// TIA Portal V15.1 export
// export: Created 2024-05-17T05:38:31.1004631Z, ExportSetting WithDefaults, DisplayName Totally Integrated Automation Portal, DisplayVersion V15.1 Update 5, DisplayName TIA Portal Openness, DisplayVersion V15.1 Update 5, DisplayName SINAMICS Startdrive Advanced, DisplayVersion V15.1, DisplayName G130, G150, S120, S150, SINAMICS MV, S210, DisplayVersion V15.1, DisplayName G110M, G120, G120C, G120D, G120P, DisplayVersion V15.1, DisplayName STEP 7 Professional, DisplayVersion V15.1 Update 5, DisplayName STEP 7 Safety, DisplayVersion V15.1, DisplayName WinCC Professional, DisplayVersion V15.1 Update 5, DisplayName SIMATIC Visualization Architect, DisplayVersion V15.1
FUNCTION_BLOCK "LProductionMode"   // FB1003, FBD
TITLE = LProductionMode
{ S7_Optimized_Access := 'FALSE' }
AUTHOR : VCC
FAMILY : Control
NAME : ProdMode
VERSION : 1.0
// ================================================================================
// This module handles all production modes for a modezone. The production modes 
// are Bypass, Empty Station, Simulation with/without part, Maintenance, Cycle 
// Stop and Production Stop.
// ================================================================================
// stored: AutoNumber false, IsIECCheckEnabled false, SetENOAutomatically False, UDAEnableTagReadback false
   VAR_INPUT
      I_BypassStartCond { ExternalAccessible := 'False'; ExternalVisible := 'False'; ExternalWritable := 'False'} : Bool;   // Start condition for Bypass mode
      I_ExtBypassReq { ExternalAccessible := 'False'; ExternalVisible := 'False'; ExternalWritable := 'False'} : Bool;   // External bypass request
      I_EmptyStnReached { ExternalAccessible := 'False'; ExternalVisible := 'False'; ExternalWritable := 'False'} : Bool;   // Empty station reached
      I_ExtEmptyStnReq { ExternalAccessible := 'False'; ExternalVisible := 'False'; ExternalWritable := 'False'} : Bool;   // External Empty station request
      I_SimWithPartStartCond { ExternalAccessible := 'False'; ExternalVisible := 'False'; ExternalWritable := 'False'} : Bool;   // Start condition for Simulation with part mode
      I_ExtSimWithPartReq { ExternalAccessible := 'False'; ExternalVisible := 'False'; ExternalWritable := 'False'} : Bool;   // External Simulation with part request
      I_SimWithoutPartStartCon { ExternalAccessible := 'False'; ExternalVisible := 'False'; ExternalWritable := 'False'} : Bool;   // Start condition for Simulation without part mode
      I_ExtSimWithoutPartReq { ExternalAccessible := 'False'; ExternalVisible := 'False'; ExternalWritable := 'False'} : Bool;   // External Simulation without part request
      I_MaintStartCond { ExternalAccessible := 'False'; ExternalVisible := 'False'; ExternalWritable := 'False'} : Bool;   // Start condition for maintenance mode
      I_ExtMaintReq { ExternalAccessible := 'False'; ExternalVisible := 'False'; ExternalWritable := 'False'} : Bool;   // External Maintenance request
      I_MaintReached { ExternalAccessible := 'False'; ExternalVisible := 'False'; ExternalWritable := 'False'} : Bool;   // Maintenance reached
      I_CycleStpBeforeReached { ExternalAccessible := 'False'; ExternalVisible := 'False'; ExternalWritable := 'False'} : Bool;   // Cycle stop before work reached
      I_ExtCycleStpBeforeReq { ExternalAccessible := 'False'; ExternalVisible := 'False'; ExternalWritable := 'False'} : Bool;   // External Cycle stop before work request
      I_CycleStpAfterReached { ExternalAccessible := 'False'; ExternalVisible := 'False'; ExternalWritable := 'False'} : Bool;   // Cycle stop after work reached
      I_ExtCycleStpAfterReq { ExternalAccessible := 'False'; ExternalVisible := 'False'; ExternalWritable := 'False'} : Bool;   // External Cycle stop after work request
      I_ProdStpReached { ExternalAccessible := 'False'; ExternalVisible := 'False'; ExternalWritable := 'False'} : Bool;   // Production mode reached
      I_ExtProdStpReq { ExternalAccessible := 'False'; ExternalVisible := 'False'; ExternalWritable := 'False'} : Bool;   // External production stop request
      I_AlarmResetPB { ExternalAccessible := 'False'; ExternalVisible := 'False'; ExternalWritable := 'False'} : Bool;   // Alarm reset pushbutton is activated
   END_VAR
   VAR_OUTPUT
      O_ProductionMode { ExternalAccessible := 'False'; ExternalVisible := 'False'; ExternalWritable := 'False'} : Word;   // Prodution Modes
      O_BypassModeSel { ExternalAccessible := 'False'; ExternalVisible := 'False'; ExternalWritable := 'False'} : Bool;   // Bypass mode selected
      O_BypassMode { ExternalAccessible := 'False'; ExternalVisible := 'False'; ExternalWritable := 'False'} : Bool;   // Bypass mode active
      O_EmptyStnModeSel { ExternalAccessible := 'False'; ExternalVisible := 'False'; ExternalWritable := 'False'} : Bool;   // Empty station mode selected
      O_EmptyStnMode { ExternalAccessible := 'False'; ExternalVisible := 'False'; ExternalWritable := 'False'} : Bool;   // Empty station mode active
      O_SimWithPartModeSel { ExternalAccessible := 'False'; ExternalVisible := 'False'; ExternalWritable := 'False'} : Bool;   // Simulation with part mode selected
      O_SimWithPartMode { ExternalAccessible := 'False'; ExternalVisible := 'False'; ExternalWritable := 'False'} : Bool;   // Simulation with part mode active
      O_SimWithoutPartModeSel { ExternalAccessible := 'False'; ExternalVisible := 'False'; ExternalWritable := 'False'} : Bool;   // Simulation without part mode selcted
      O_SimWithoutPartMode { ExternalAccessible := 'False'; ExternalVisible := 'False'; ExternalWritable := 'False'} : Bool;   // Simulation without part mode active
      O_MaintModeSel { ExternalAccessible := 'False'; ExternalVisible := 'False'; ExternalWritable := 'False'} : Bool;   // Maintenance mode selected
      O_MaintMode { ExternalAccessible := 'False'; ExternalVisible := 'False'; ExternalWritable := 'False'} : Bool;   // Maintenance mode active
      O_CycleStpBeforeModeSel { ExternalAccessible := 'False'; ExternalVisible := 'False'; ExternalWritable := 'False'} : Bool;   // Cycle stop before mode selected
      O_CycleStpBeforeMode { ExternalAccessible := 'False'; ExternalVisible := 'False'; ExternalWritable := 'False'} : Bool;   // Cycle stop before mode active
      O_CycleStpAfterModeSel { ExternalAccessible := 'False'; ExternalVisible := 'False'; ExternalWritable := 'False'} : Bool;   // Cycle stop after mode selected
      O_CycleStpAfterMode { ExternalAccessible := 'False'; ExternalVisible := 'False'; ExternalWritable := 'False'} : Bool;   // Cycle stop after mode active
      O_ProdStpModeSel { ExternalAccessible := 'False'; ExternalVisible := 'False'; ExternalWritable := 'False'} : Bool;   // Production mode selected
      O_ProdStpMode { ExternalAccessible := 'False'; ExternalVisible := 'False'; ExternalWritable := 'False'} : Bool;   // Production mode active
      O_AnyProdModeSel { ExternalAccessible := 'False'; ExternalVisible := 'False'; ExternalWritable := 'False'} : Bool;   // Any production mode selected
      O_AnyProdModeActive { ExternalAccessible := 'False'; ExternalVisible := 'False'; ExternalWritable := 'False'} : Bool;   // Any production mode active
      O_AlarmABCondition { ExternalAccessible := 'False'; ExternalVisible := 'False'; ExternalWritable := 'False'} : Bool;   // Alarm AB condition
      O_AlarmA { ExternalAccessible := 'False'; ExternalVisible := 'False'; ExternalWritable := 'False'} : Bool;   // Alarms A
      O_AlarmB { ExternalAccessible := 'False'; ExternalVisible := 'False'; ExternalWritable := 'False'} : Bool;   // Alarms B
      O_AlarmC { ExternalAccessible := 'False'; ExternalVisible := 'False'; ExternalWritable := 'False'} : Bool;   // Alarms C
      O_AlarmD { ExternalAccessible := 'False'; ExternalVisible := 'False'; ExternalWritable := 'False'} : Bool;   // Alarms D
      H_AlarmWord { ExternalAccessible := 'False'; ExternalVisible := 'False'; ExternalWritable := 'False'} : DWord;   // Alarm Word
   END_VAR
   VAR_IN_OUT
      IO_Modes : "Modes";
   END_VAR
   VAR DB_SPECIFIC
      AB_SimWithPartAlm { ExternalAccessible := 'False'; ExternalVisible := 'False'; ExternalWritable := 'False'} : Bool;   // Condition missing for simulation with part
      AB_SimWithoutPartAlm { ExternalAccessible := 'False'; ExternalVisible := 'False'; ExternalWritable := 'False'} : Bool;   // Condition missing for simulation without part
      AD_EmptyStnSelected { ExternalAccessible := 'False'; ExternalVisible := 'False'; ExternalWritable := 'False'} : Bool;   // Empty station is selected
      AD_BypassSelected { ExternalAccessible := 'False'; ExternalVisible := 'False'; ExternalWritable := 'False'} : Bool;   // Bypass is selected
      AD_SimWithPartSelected { ExternalAccessible := 'False'; ExternalVisible := 'False'; ExternalWritable := 'False'} : Bool;   // Simulation with part is selected
      AD_SimWithoutPartSel { ExternalAccessible := 'False'; ExternalVisible := 'False'; ExternalWritable := 'False'} : Bool;   // Simulation without part is selected
      AD_MaintSelected { ExternalAccessible := 'False'; ExternalVisible := 'False'; ExternalWritable := 'False'} : Bool;   // Maintenance is selected
      AD_ProdStpSelected { ExternalAccessible := 'False'; ExternalVisible := 'False'; ExternalWritable := 'False'} : Bool;   // Production stop is selected
      AD_CycleStpBeforeSel { ExternalAccessible := 'False'; ExternalVisible := 'False'; ExternalWritable := 'False'} : Bool;   // Cycle stop before is selected
      AD_CycleStpAfterSelected { ExternalAccessible := 'False'; ExternalVisible := 'False'; ExternalWritable := 'False'} : Bool;   // Cycle stop after is selected
      H_HMIProdModeCmd : Word;   // Production mode commands from HMI
      H_Anim : Word;   // Animation
      H_Anim2 : Word;   // Animation word 2
      SimWithPartAlmCond { ExternalAccessible := 'False'; ExternalVisible := 'False'; ExternalWritable := 'False'} : Bool;   // Alarm condition for Simulation with part
      SimWithoutPartAlmCond { ExternalAccessible := 'False'; ExternalVisible := 'False'; ExternalWritable := 'False'} : Bool;   // Alarm condition for Simulation without part
      HMIBypassReq { ExternalAccessible := 'False'; ExternalVisible := 'False'; ExternalWritable := 'False'} : Bool;   // Bypass selected on HMI
      HMIEmptyStnReq { ExternalAccessible := 'False'; ExternalVisible := 'False'; ExternalWritable := 'False'} : Bool;   // Empty station selected on HMI
      HMISimWithPartReq { ExternalAccessible := 'False'; ExternalVisible := 'False'; ExternalWritable := 'False'} : Bool;   // Simulation with part selected on HMI
      HMISimWithoutPartReq { ExternalAccessible := 'False'; ExternalVisible := 'False'; ExternalWritable := 'False'} : Bool;   // Simulation without part selected on HMI
      HMIMaintReq { ExternalAccessible := 'False'; ExternalVisible := 'False'; ExternalWritable := 'False'} : Bool;   // Maintenance selected on HMI
      HMICycleStpBeforeReq { ExternalAccessible := 'False'; ExternalVisible := 'False'; ExternalWritable := 'False'} : Bool;   // Cycle stop before work selected on HMI
      HMICycleStpAfterReq { ExternalAccessible := 'False'; ExternalVisible := 'False'; ExternalWritable := 'False'} : Bool;   // Cycle stop after work selected on HMI
      HMIProdStpReq { ExternalAccessible := 'False'; ExternalVisible := 'False'; ExternalWritable := 'False'} : Bool;   // Production mode selected on HMI
      EmptyStnActive { ExternalAccessible := 'False'; ExternalVisible := 'False'; ExternalWritable := 'False'} : Bool;   // Empty station is active
      BypassActive { ExternalAccessible := 'False'; ExternalVisible := 'False'; ExternalWritable := 'False'} : Bool;   // Bypass is active
      SimWithPartActive { ExternalAccessible := 'False'; ExternalVisible := 'False'; ExternalWritable := 'False'} : Bool;   // Simulation with part is active
      SimWithoutPartActive { ExternalAccessible := 'False'; ExternalVisible := 'False'; ExternalWritable := 'False'} : Bool;   // Simulation without part is active
      SimDeactivate { ExternalAccessible := 'False'; ExternalVisible := 'False'; ExternalWritable := 'False'} : Bool;   // Deactivate simulation
      MaintActive { ExternalAccessible := 'False'; ExternalVisible := 'False'; ExternalWritable := 'False'} : Bool;   // Maintenance is active
      ProdStpActive { ExternalAccessible := 'False'; ExternalVisible := 'False'; ExternalWritable := 'False'} : Bool;   // Production stop is active
      CycleStpBeforeActive { ExternalAccessible := 'False'; ExternalVisible := 'False'; ExternalWritable := 'False'} : Bool;   // Cycle stop before is active
      CycleStpAfterActive { ExternalAccessible := 'False'; ExternalVisible := 'False'; ExternalWritable := 'False'} : Bool;   // Cycle stop after is active
      PulseSimWithPartSel { ExternalAccessible := 'False'; ExternalVisible := 'False'; ExternalWritable := 'False'} : Bool;   // Pulse simulation with part selected
      PulseSimWithoutPartSel { ExternalAccessible := 'False'; ExternalVisible := 'False'; ExternalWritable := 'False'} : Bool;   // Pulse simulation without part selected
      TmpMaintReqOn { ExternalAccessible := 'False'; ExternalVisible := 'False'; ExternalWritable := 'False'} : Bool;   // Temporary request on
      TmpBypassReqOn { ExternalAccessible := 'False'; ExternalVisible := 'False'; ExternalWritable := 'False'} : Bool;   // Temporary request on
      TmpEmptyStnReqOn { ExternalAccessible := 'False'; ExternalVisible := 'False'; ExternalWritable := 'False'} : Bool;   // Temporary request on
      TmpProdStpReqOn { ExternalAccessible := 'False'; ExternalVisible := 'False'; ExternalWritable := 'False'} : Bool;   // Temporary request on
      AlarmA { ExternalAccessible := 'False'; ExternalVisible := 'False'; ExternalWritable := 'False'} : Bool;   // Alarm A active in the FB
      AlarmB { ExternalAccessible := 'False'; ExternalVisible := 'False'; ExternalWritable := 'False'} : Bool;   // Alarm B active in the FB
      AlarmC { ExternalAccessible := 'False'; ExternalVisible := 'False'; ExternalWritable := 'False'} : Bool;   // Alarm C active in the FB
      AlarmD { ExternalAccessible := 'False'; ExternalVisible := 'False'; ExternalWritable := 'False'} : Bool;   // Alarm D active in the FB
      TmpSimWithoutPartReqOn { ExternalAccessible := 'False'; ExternalVisible := 'False'; ExternalWritable := 'False'} : Bool;   // Temporary request on
      TmpSimWithPartReqOn { ExternalAccessible := 'False'; ExternalVisible := 'False'; ExternalWritable := 'False'} : Bool;   // Temporary request on
   END_VAR
   VAR
      ToggleBypassReq { ExternalAccessible := 'False'; ExternalVisible := 'False'; ExternalWritable := 'False'; S7_SetPoint := 'True'} : "LToggle";
      ToggleEmptyStnReq { ExternalAccessible := 'False'; ExternalVisible := 'False'; ExternalWritable := 'False'; S7_SetPoint := 'True'} : "LToggle";
      ToggleSimWithPartReq { ExternalAccessible := 'False'; ExternalVisible := 'False'; ExternalWritable := 'False'; S7_SetPoint := 'True'} : "LToggle";
      ToggleMaintReq { ExternalAccessible := 'False'; ExternalVisible := 'False'; ExternalWritable := 'False'; S7_SetPoint := 'True'} : "LToggle";
      ToggleCycleStpBeforeReq { ExternalAccessible := 'False'; ExternalVisible := 'False'; ExternalWritable := 'False'; S7_SetPoint := 'True'} : "LToggle";
      ToggleCycleStpAfterReq { ExternalAccessible := 'False'; ExternalVisible := 'False'; ExternalWritable := 'False'; S7_SetPoint := 'True'} : "LToggle";
      ToggleProsStpReq { ExternalAccessible := 'False'; ExternalVisible := 'False'; ExternalWritable := 'False'; S7_SetPoint := 'True'} : "LToggle";
      ToggleSimWithoutPartReq { ExternalAccessible := 'False'; ExternalVisible := 'False'; ExternalWritable := 'False'; S7_SetPoint := 'True'} : "LToggle";
   END_VAR
   VAR_TEMP   // added for the SCL form of the ladder/FBD networks
      _w1 : Bool;
   END_VAR
BEGIN

REGION Network 1: **** 1 - Inputs **** Extract the production modes from HMI
   // Extract the production modes from HMI
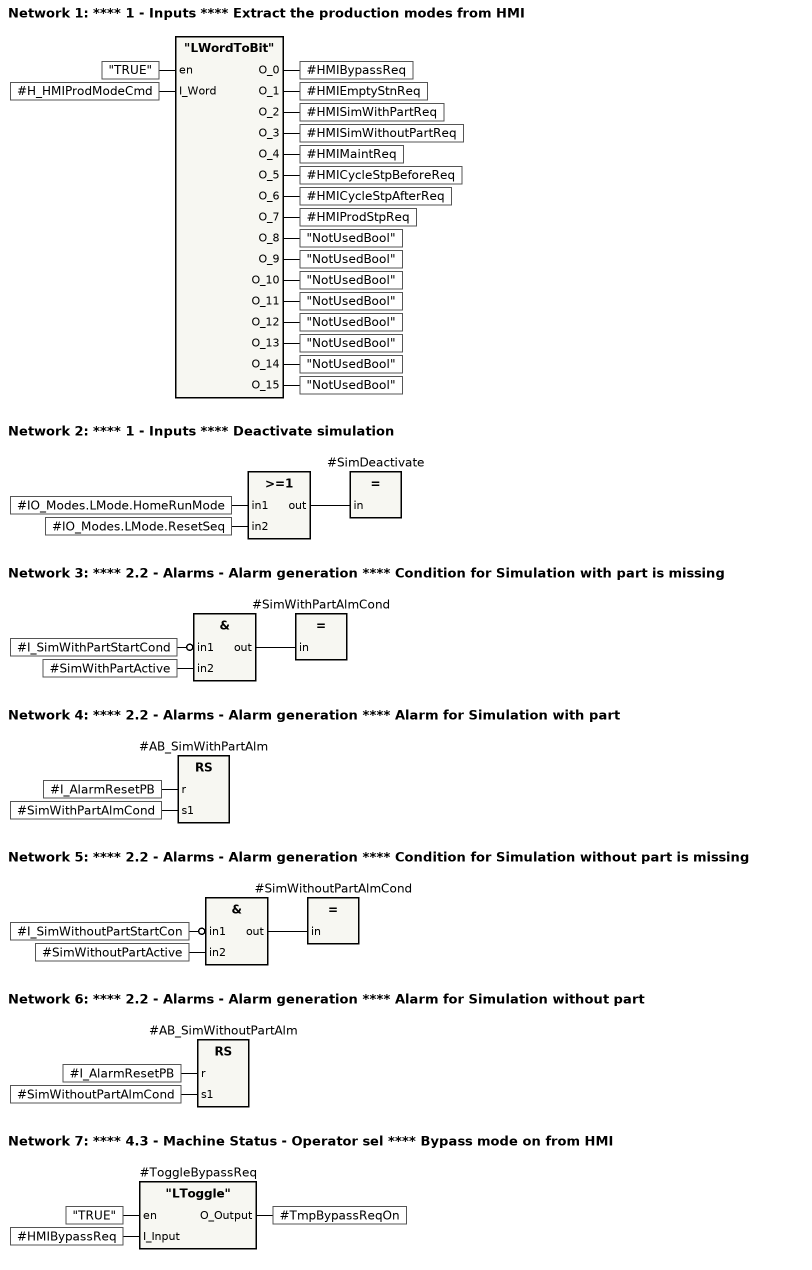
   IF "TRUE" THEN
       "LWordToBit"(I_Word := #H_HMIProdModeCmd,
                    O_0 => #HMIBypassReq,
                    O_1 => #HMIEmptyStnReq,
                    O_2 => #HMISimWithPartReq,
                    O_3 => #HMISimWithoutPartReq,
                    O_4 => #HMIMaintReq,
                    O_5 => #HMICycleStpBeforeReq,
                    O_6 => #HMICycleStpAfterReq,
                    O_7 => #HMIProdStpReq,
                    O_8 => "NotUsedBool",
                    O_9 => "NotUsedBool",
                    O_10 => "NotUsedBool",
                    O_11 => "NotUsedBool",
                    O_12 => "NotUsedBool",
                    O_13 => "NotUsedBool",
                    O_14 => "NotUsedBool",
                    O_15 => "NotUsedBool");
   END_IF;
END_REGION

REGION Network 2: **** 1 - Inputs **** Deactivate simulation
   #SimDeactivate := #IO_Modes.LMode.HomeRunMode OR #IO_Modes.LMode.ResetSeq;
END_REGION

REGION Network 3: **** 2.2 - Alarms - Alarm generation **** Condition for Simulation with part is missing
   // Condition for Simulation with part is missing
   #SimWithPartAlmCond := NOT #I_SimWithPartStartCond AND #SimWithPartActive;
END_REGION

REGION Network 4: **** 2.2 - Alarms - Alarm generation **** Alarm for Simulation with part
   // Alarm for Simulation with part
   IF #I_AlarmResetPB THEN
       #AB_SimWithPartAlm := FALSE;   // RS flip-flop
   END_IF;
   IF #SimWithPartAlmCond THEN #AB_SimWithPartAlm := TRUE; END_IF;
END_REGION

REGION Network 5: **** 2.2 - Alarms - Alarm generation **** Condition for Simulation without part is missing
   // Condition for Simulation without part is missing
   #SimWithoutPartAlmCond := NOT #I_SimWithoutPartStartCon AND #SimWithoutPartActive;
END_REGION

REGION Network 6: **** 2.2 - Alarms - Alarm generation **** Alarm for Simulation without part
   // Alarm for Simulation without part
   IF #I_AlarmResetPB THEN
       #AB_SimWithoutPartAlm := FALSE;   // RS flip-flop
   END_IF;
   IF #SimWithoutPartAlmCond THEN #AB_SimWithoutPartAlm := TRUE; END_IF;
END_REGION

REGION Network 7: **** 4.3 - Machine Status - Operator sel **** Bypass mode on from HMI
   // Bypass mode on from HMI
   IF "TRUE" THEN
       #ToggleBypassReq(I_Input := #HMIBypassReq, O_Output => #TmpBypassReqOn);   // "LToggle"
   END_IF;
END_REGION

REGION Network 8: **** 4.3 - Machine Status - Operator sel **** Bypass mode is selected
   // Bypass mode is selected
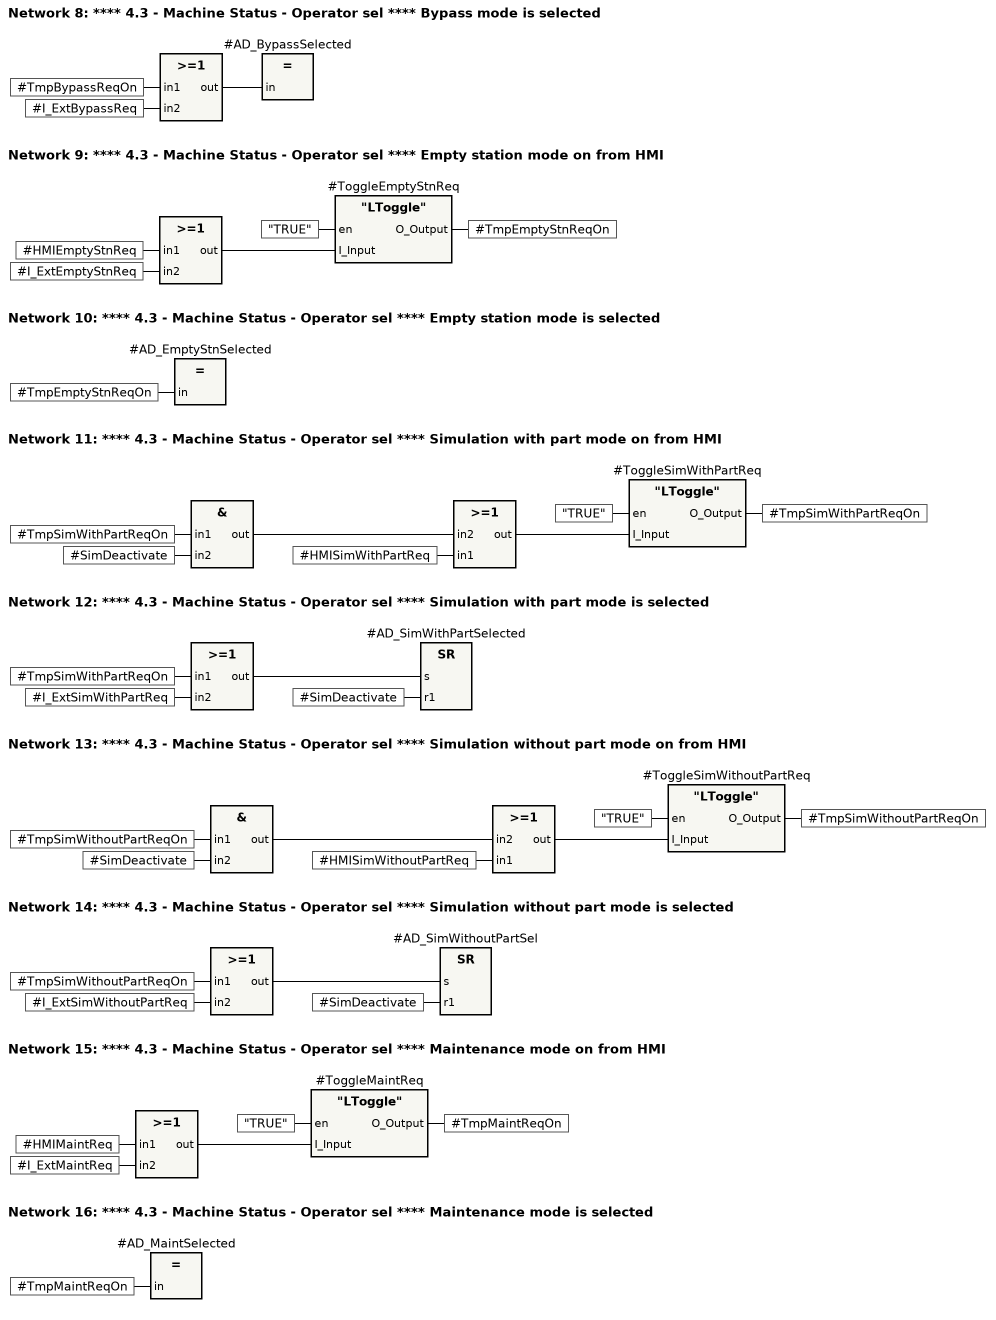
   #AD_BypassSelected := #TmpBypassReqOn OR #I_ExtBypassReq;
END_REGION

REGION Network 9: **** 4.3 - Machine Status - Operator sel **** Empty station mode on from HMI
   // Empty station mode on from HMI
   IF "TRUE" THEN
       #ToggleEmptyStnReq(I_Input := #HMIEmptyStnReq OR #I_ExtEmptyStnReq, O_Output => #TmpEmptyStnReqOn);   // "LToggle"
   END_IF;
END_REGION

REGION Network 10: **** 4.3 - Machine Status - Operator sel **** Empty station mode is selected
   // Empty station mode is selected
   #AD_EmptyStnSelected := #TmpEmptyStnReqOn;
END_REGION

REGION Network 11: **** 4.3 - Machine Status - Operator sel **** Simulation with part mode on from HMI
   // Simulation with part mode on from HMI
   IF "TRUE" THEN
       #ToggleSimWithPartReq(I_Input := (#TmpSimWithPartReqOn AND #SimDeactivate) OR #HMISimWithPartReq,   // "LToggle"
                             O_Output => #TmpSimWithPartReqOn);
   END_IF;
END_REGION

REGION Network 12: **** 4.3 - Machine Status - Operator sel **** Simulation with part mode is selected
   // Simulation with part mode is selected
   IF #TmpSimWithPartReqOn OR #I_ExtSimWithPartReq THEN
       #AD_SimWithPartSelected := TRUE;   // SR flip-flop
   END_IF;
   IF #SimDeactivate THEN #AD_SimWithPartSelected := FALSE; END_IF;
END_REGION

REGION Network 13: **** 4.3 - Machine Status - Operator sel **** Simulation without part mode on from HMI
   // Simulation without part mode on from HMI
   IF "TRUE" THEN
       #ToggleSimWithoutPartReq(I_Input := (#TmpSimWithoutPartReqOn AND #SimDeactivate) OR #HMISimWithoutPartReq,   // "LToggle"
                               O_Output => #TmpSimWithoutPartReqOn);
   END_IF;
END_REGION

REGION Network 14: **** 4.3 - Machine Status - Operator sel **** Simulation without part mode is selected
   // Simulation without part mode is selected
   IF #TmpSimWithoutPartReqOn OR #I_ExtSimWithoutPartReq THEN
       #AD_SimWithoutPartSel := TRUE;   // SR flip-flop
   END_IF;
   IF #SimDeactivate THEN #AD_SimWithoutPartSel := FALSE; END_IF;
END_REGION

REGION Network 15: **** 4.3 - Machine Status - Operator sel **** Maintenance mode on from HMI
   // Maintenance mode on from HMI
   IF "TRUE" THEN
       #ToggleMaintReq(I_Input := #HMIMaintReq OR #I_ExtMaintReq, O_Output => #TmpMaintReqOn);   // "LToggle"
   END_IF;
END_REGION

REGION Network 16: **** 4.3 - Machine Status - Operator sel **** Maintenance mode is selected
   // Maintenance mode is selected
   #AD_MaintSelected := #TmpMaintReqOn;
END_REGION

REGION Network 17: **** 4.3 - Machine Status - Operator sel **** Cycle stop before mode is selected
   // Cycle stop before mode is selected
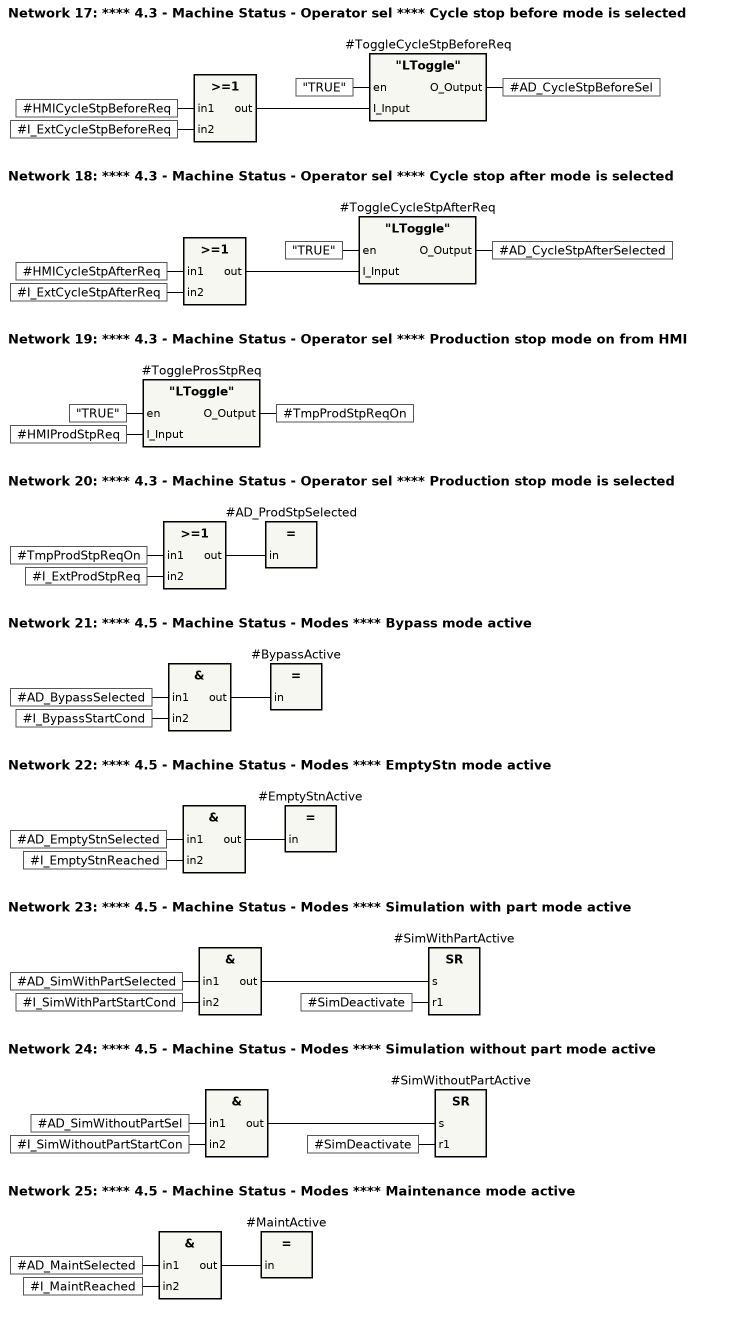
   IF "TRUE" THEN
       #ToggleCycleStpBeforeReq(I_Input := #HMICycleStpBeforeReq OR #I_ExtCycleStpBeforeReq,   // "LToggle"
                               O_Output => #AD_CycleStpBeforeSel);
   END_IF;
END_REGION

REGION Network 18: **** 4.3 - Machine Status - Operator sel **** Cycle stop after mode is selected
   // Cycle stop after mode is selected
   IF "TRUE" THEN
       #ToggleCycleStpAfterReq(I_Input := #HMICycleStpAfterReq OR #I_ExtCycleStpAfterReq,   // "LToggle"
                               O_Output => #AD_CycleStpAfterSelected);
   END_IF;
END_REGION

REGION Network 19: **** 4.3 - Machine Status - Operator sel **** Production stop mode on from HMI
   // Production stop mode on from HMI
   IF "TRUE" THEN
       #ToggleProsStpReq(I_Input := #HMIProdStpReq, O_Output => #TmpProdStpReqOn);   // "LToggle"
   END_IF;
END_REGION

REGION Network 20: **** 4.3 - Machine Status - Operator sel **** Production stop mode is selected
   // Production stop mode is selected
   #AD_ProdStpSelected := #TmpProdStpReqOn OR #I_ExtProdStpReq;
END_REGION

REGION Network 21: **** 4.5 - Machine Status - Modes **** Bypass mode active
   // Bypass mode active
   #BypassActive := #AD_BypassSelected AND #I_BypassStartCond;
END_REGION

REGION Network 22: **** 4.5 - Machine Status - Modes **** EmptyStn mode active
   // EmptyStn mode active
   #EmptyStnActive := #AD_EmptyStnSelected AND #I_EmptyStnReached;
END_REGION

REGION Network 23: **** 4.5 - Machine Status - Modes **** Simulation with part mode active
   // Simulation with part mode active
   IF #AD_SimWithPartSelected AND #I_SimWithPartStartCond THEN
       #SimWithPartActive := TRUE;   // SR flip-flop
   END_IF;
   IF #SimDeactivate THEN #SimWithPartActive := FALSE; END_IF;
END_REGION

REGION Network 24: **** 4.5 - Machine Status - Modes **** Simulation without part mode active
   // Simulation without part mode active
   IF #AD_SimWithoutPartSel AND #I_SimWithoutPartStartCon THEN
       #SimWithoutPartActive := TRUE;   // SR flip-flop
   END_IF;
   IF #SimDeactivate THEN #SimWithoutPartActive := FALSE; END_IF;
END_REGION

REGION Network 25: **** 4.5 - Machine Status - Modes **** Maintenance mode active
   // Maintenance mode active
   #MaintActive := #AD_MaintSelected AND #I_MaintReached;
END_REGION

REGION Network 26: **** 4.5 - Machine Status - Modes **** Cycle Stop Before mode active
   // Cycle Stop Before mode active
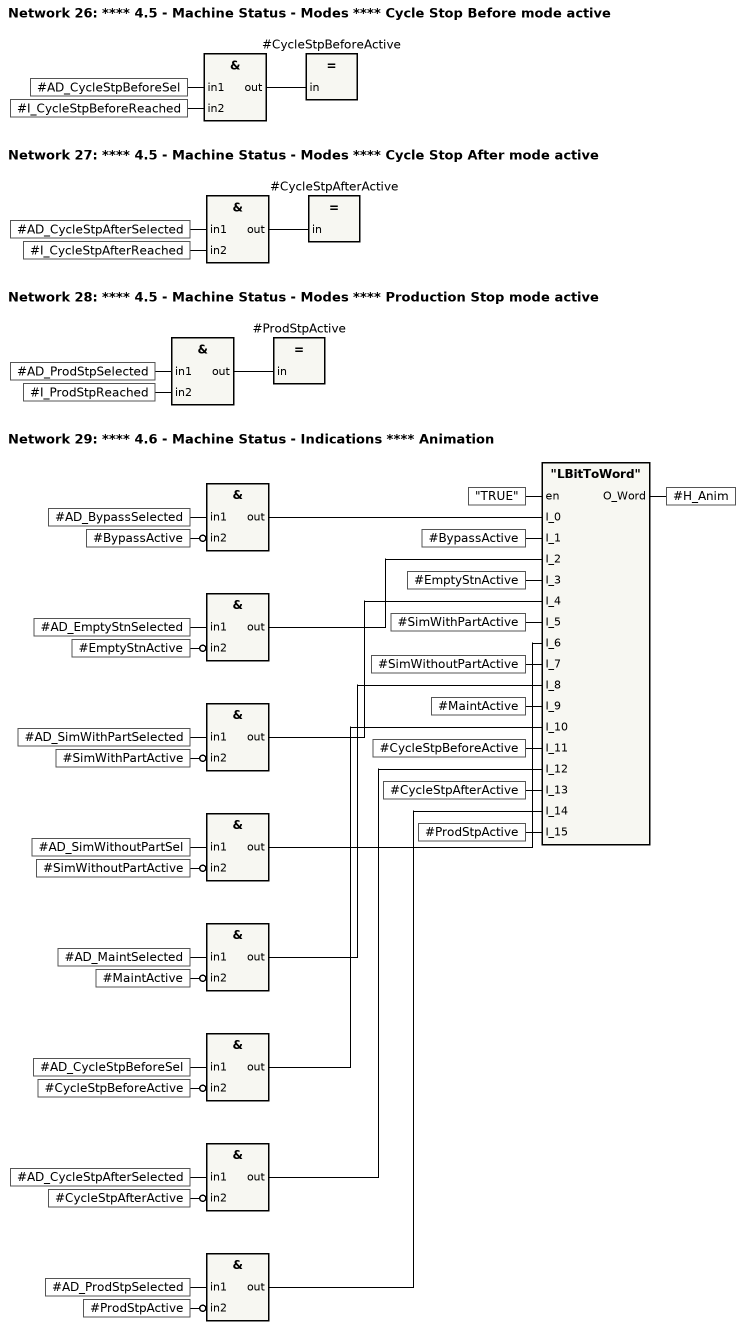
   #CycleStpBeforeActive := #AD_CycleStpBeforeSel AND #I_CycleStpBeforeReached;
END_REGION

REGION Network 27: **** 4.5 - Machine Status - Modes **** Cycle Stop After mode active
   // Cycle Stop After mode active
   #CycleStpAfterActive := #AD_CycleStpAfterSelected AND #I_CycleStpAfterReached;
END_REGION

REGION Network 28: **** 4.5 - Machine Status - Modes **** Production Stop mode active
   // Production Stop mode active
   #ProdStpActive := #AD_ProdStpSelected AND #I_ProdStpReached;
END_REGION

REGION Network 29: **** 4.6 - Machine Status - Indications **** Animation
   // Animation
   IF "TRUE" THEN
       "LBitToWord"(I_0 := #AD_BypassSelected AND NOT #BypassActive,
                    I_1 := #BypassActive,
                    I_2 := #AD_EmptyStnSelected AND NOT #EmptyStnActive,
                    I_3 := #EmptyStnActive,
                    I_4 := #AD_SimWithPartSelected AND NOT #SimWithPartActive,
                    I_5 := #SimWithPartActive,
                    I_6 := #AD_SimWithoutPartSel AND NOT #SimWithoutPartActive,
                    I_7 := #SimWithoutPartActive,
                    I_8 := #AD_MaintSelected AND NOT #MaintActive,
                    I_9 := #MaintActive,
                    I_10 := #AD_CycleStpBeforeSel AND NOT #CycleStpBeforeActive,
                    I_11 := #CycleStpBeforeActive,
                    I_12 := #AD_CycleStpAfterSelected AND NOT #CycleStpAfterActive,
                    I_13 := #CycleStpAfterActive,
                    I_14 := #AD_ProdStpSelected AND NOT #ProdStpActive,
                    I_15 := #ProdStpActive,
                    O_Word => #H_Anim);
   END_IF;
END_REGION

REGION Network 30: **** 4.6 - Machine Status - Indications **** Animation2
   // Animation word 2
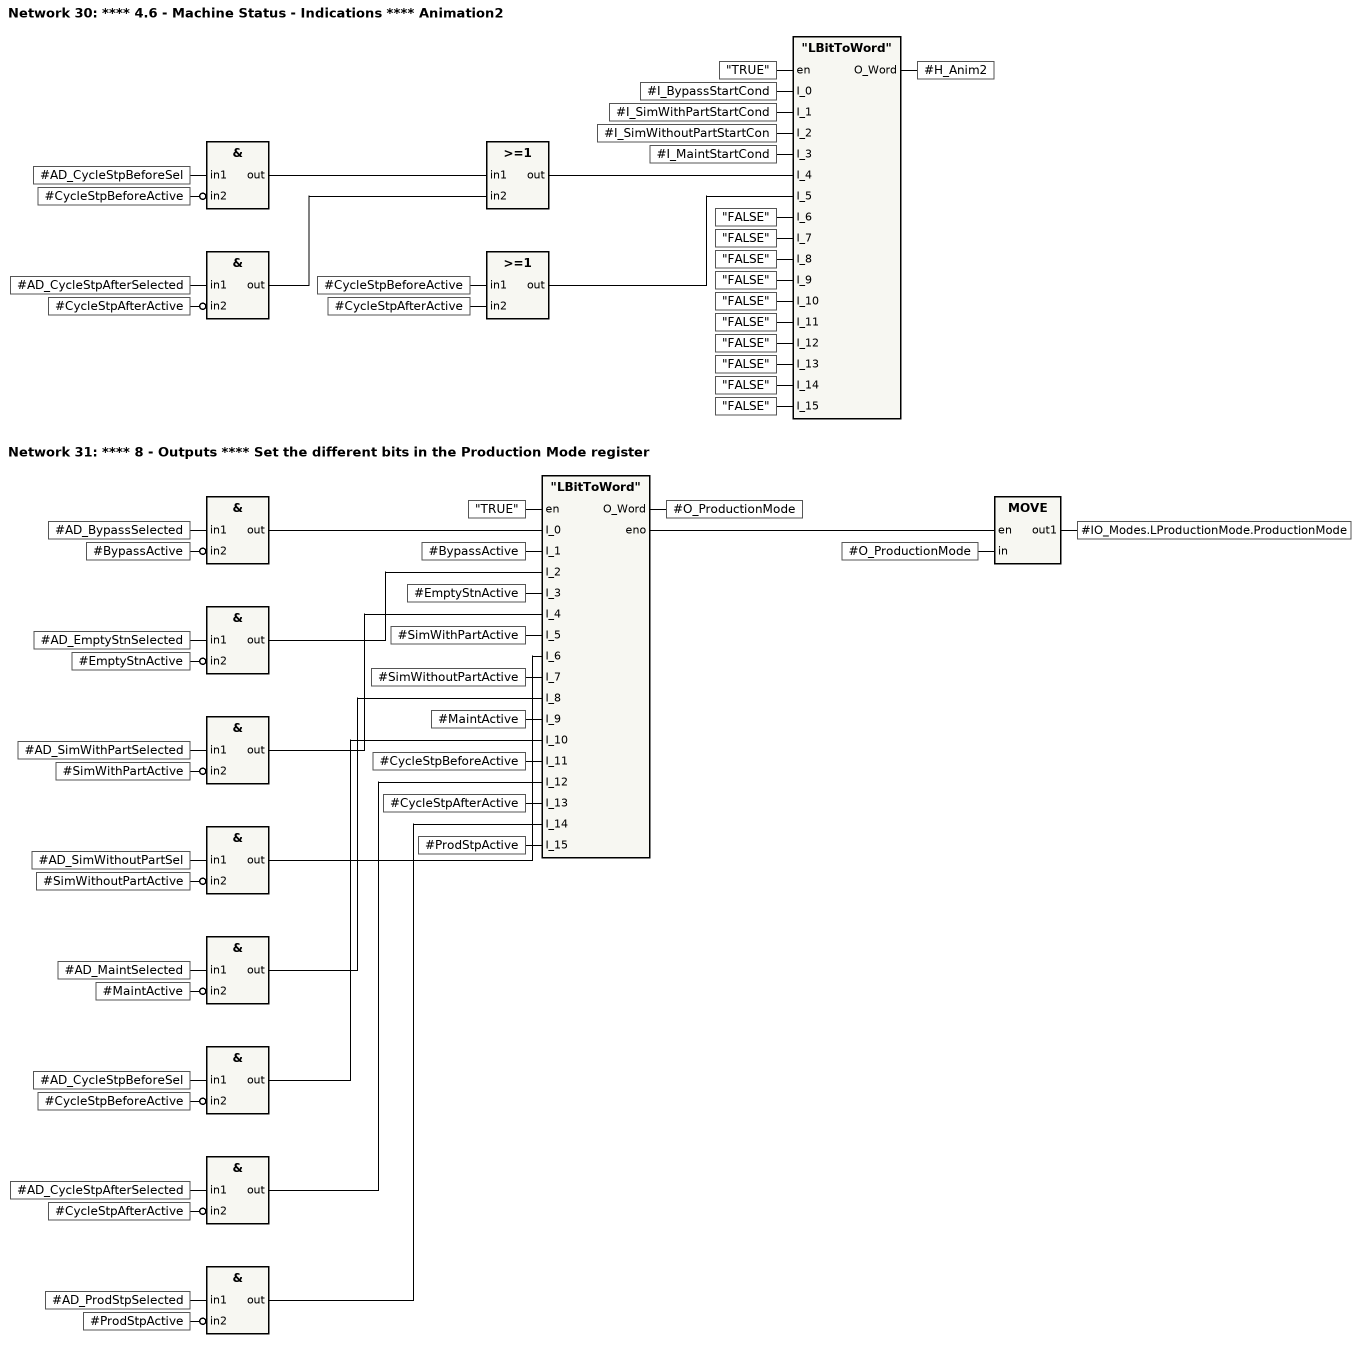
   IF "TRUE" THEN
       "LBitToWord"(I_0 := #I_BypassStartCond,
                    I_1 := #I_SimWithPartStartCond,
                    I_2 := #I_SimWithoutPartStartCon,
                    I_3 := #I_MaintStartCond,
                    I_4 := (#AD_CycleStpBeforeSel AND NOT #CycleStpBeforeActive) OR (#AD_CycleStpAfterSelected AND NOT #CycleStpAfterActive),
                    I_5 := #CycleStpBeforeActive OR #CycleStpAfterActive,
                    I_6 := "FALSE",
                    I_7 := "FALSE",
                    I_8 := "FALSE",
                    I_9 := "FALSE",
                    I_10 := "FALSE",
                    I_11 := "FALSE",
                    I_12 := "FALSE",
                    I_13 := "FALSE",
                    I_14 := "FALSE",
                    I_15 := "FALSE",
                    O_Word => #H_Anim2);
   END_IF;
END_REGION

REGION Network 31: **** 8 - Outputs **** Set the different bits in the Production Mode register
   // Set the different bits in the Production Mode register
   "LBitToWord"(EN := "TRUE",
                I_0 := #AD_BypassSelected AND NOT #BypassActive,
                I_1 := #BypassActive,
                I_2 := #AD_EmptyStnSelected AND NOT #EmptyStnActive,
                I_3 := #EmptyStnActive,
                I_4 := #AD_SimWithPartSelected AND NOT #SimWithPartActive,
                I_5 := #SimWithPartActive,
                I_6 := #AD_SimWithoutPartSel AND NOT #SimWithoutPartActive,
                I_7 := #SimWithoutPartActive,
                I_8 := #AD_MaintSelected AND NOT #MaintActive,
                I_9 := #MaintActive,
                I_10 := #AD_CycleStpBeforeSel AND NOT #CycleStpBeforeActive,
                I_11 := #CycleStpBeforeActive,
                I_12 := #AD_CycleStpAfterSelected AND NOT #CycleStpAfterActive,
                I_13 := #CycleStpAfterActive,
                I_14 := #AD_ProdStpSelected AND NOT #ProdStpActive,
                I_15 := #ProdStpActive,
                O_Word => #O_ProductionMode,
                ENO => #_w1);
   IF #_w1 THEN #IO_Modes.LProductionMode.ProductionMode := #O_ProductionMode; END_IF;
END_REGION

REGION Network 32: **** 8 - Outputs **** Bypass mode selected
   // Bypass mode selected
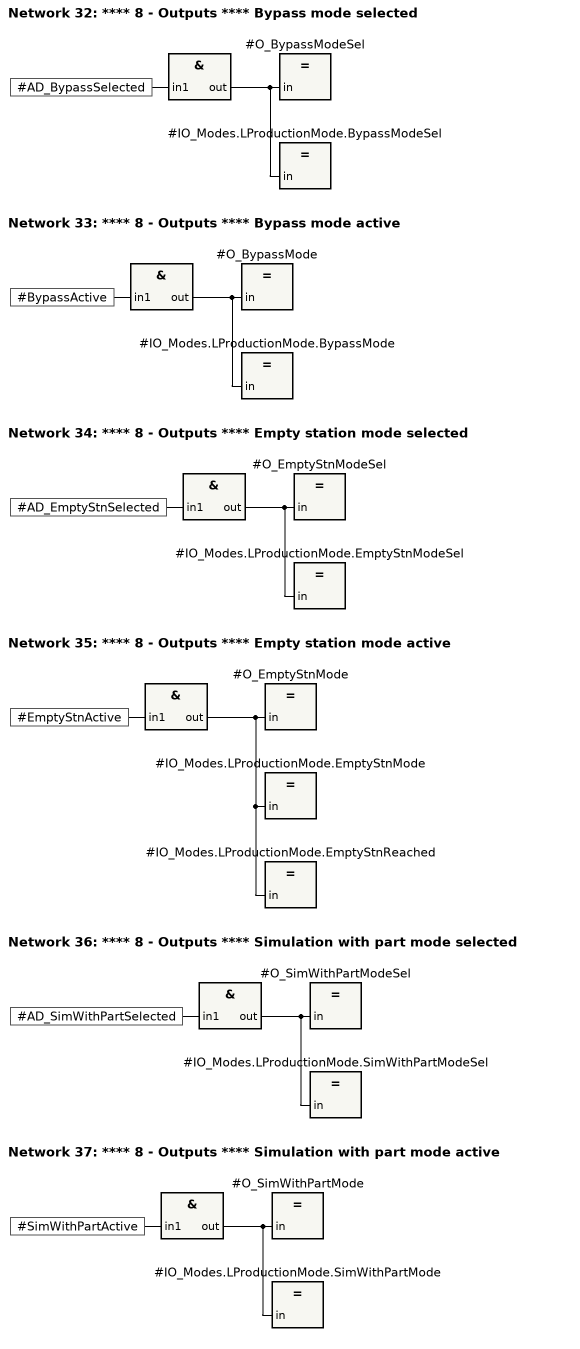
   #O_BypassModeSel := #AD_BypassSelected;
   #IO_Modes.LProductionMode.BypassModeSel := #AD_BypassSelected;
END_REGION

REGION Network 33: **** 8 - Outputs **** Bypass mode active
   // Bypass mode active
   #O_BypassMode := #BypassActive;
   #IO_Modes.LProductionMode.BypassMode := #BypassActive;
END_REGION

REGION Network 34: **** 8 - Outputs **** Empty station mode selected
   // Empty station mode selected
   #O_EmptyStnModeSel := #AD_EmptyStnSelected;
   #IO_Modes.LProductionMode.EmptyStnModeSel := #AD_EmptyStnSelected;
END_REGION

REGION Network 35: **** 8 - Outputs **** Empty station mode active
   // Empty station mode active
   #O_EmptyStnMode := #EmptyStnActive;
   #IO_Modes.LProductionMode.EmptyStnMode := #EmptyStnActive;
   #IO_Modes.LProductionMode.EmptyStnReached := #EmptyStnActive;
END_REGION

REGION Network 36: **** 8 - Outputs **** Simulation with part mode selected
   // Simulation with part mode selected
   #O_SimWithPartModeSel := #AD_SimWithPartSelected;
   #IO_Modes.LProductionMode.SimWithPartModeSel := #AD_SimWithPartSelected;
END_REGION

REGION Network 37: **** 8 - Outputs **** Simulation with part mode active
   // Simulation with part mode active
   #O_SimWithPartMode := #SimWithPartActive;
   #IO_Modes.LProductionMode.SimWithPartMode := #SimWithPartActive;
END_REGION

REGION Network 38: **** 8 - Outputs **** Simulation without part mode selected
   // Simulation without part mode selected
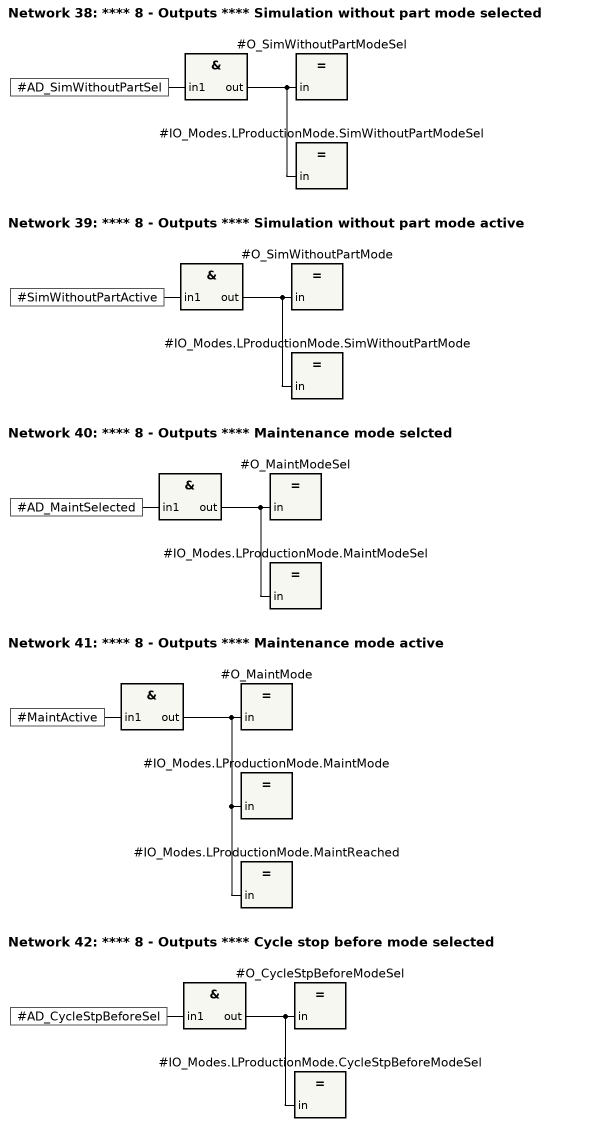
   #O_SimWithoutPartModeSel := #AD_SimWithoutPartSel;
   #IO_Modes.LProductionMode.SimWithoutPartModeSel := #AD_SimWithoutPartSel;
END_REGION

REGION Network 39: **** 8 - Outputs **** Simulation without part mode active
   // Simulation without part mode active
   #O_SimWithoutPartMode := #SimWithoutPartActive;
   #IO_Modes.LProductionMode.SimWithoutPartMode := #SimWithoutPartActive;
END_REGION

REGION Network 40: **** 8 - Outputs **** Maintenance mode selcted
   // Maintenance mode selcted
   #O_MaintModeSel := #AD_MaintSelected;
   #IO_Modes.LProductionMode.MaintModeSel := #AD_MaintSelected;
END_REGION

REGION Network 41: **** 8 - Outputs **** Maintenance mode active
   // Maintenance mode active
   #O_MaintMode := #MaintActive;
   #IO_Modes.LProductionMode.MaintMode := #MaintActive;
   #IO_Modes.LProductionMode.MaintReached := #MaintActive;
END_REGION

REGION Network 42: **** 8 - Outputs **** Cycle stop before mode selected
   // Cycle stop before mode selected
   #O_CycleStpBeforeModeSel := #AD_CycleStpBeforeSel;
   #IO_Modes.LProductionMode.CycleStpBeforeModeSel := #AD_CycleStpBeforeSel;
END_REGION

REGION Network 43: **** 8 - Outputs **** Cycle stop before mode active
   // Cycle stop before mode active
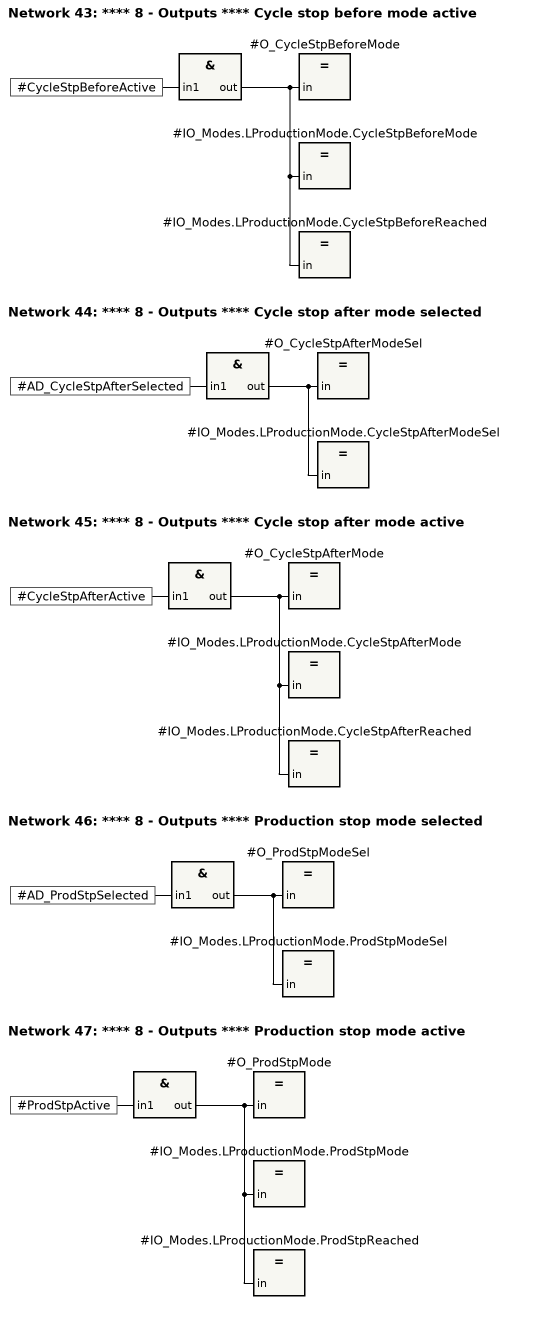
   #O_CycleStpBeforeMode := #CycleStpBeforeActive;
   #IO_Modes.LProductionMode.CycleStpBeforeMode := #CycleStpBeforeActive;
   #IO_Modes.LProductionMode.CycleStpBeforeReached := #CycleStpBeforeActive;
END_REGION

REGION Network 44: **** 8 - Outputs **** Cycle stop after mode selected
   // Cycle stop after mode selected
   #O_CycleStpAfterModeSel := #AD_CycleStpAfterSelected;
   #IO_Modes.LProductionMode.CycleStpAfterModeSel := #AD_CycleStpAfterSelected;
END_REGION

REGION Network 45: **** 8 - Outputs **** Cycle stop after mode active
   // Cycle stop after mode active
   #O_CycleStpAfterMode := #CycleStpAfterActive;
   #IO_Modes.LProductionMode.CycleStpAfterMode := #CycleStpAfterActive;
   #IO_Modes.LProductionMode.CycleStpAfterReached := #CycleStpAfterActive;
END_REGION

REGION Network 46: **** 8 - Outputs **** Production stop mode selected
   // Production stop mode selected
   #O_ProdStpModeSel := #AD_ProdStpSelected;
   #IO_Modes.LProductionMode.ProdStpModeSel := #AD_ProdStpSelected;
END_REGION

REGION Network 47: **** 8 - Outputs **** Production stop mode active
   // Production stop mode active
   #O_ProdStpMode := #ProdStpActive;
   #IO_Modes.LProductionMode.ProdStpMode := #ProdStpActive;
   #IO_Modes.LProductionMode.ProdStpReached := #ProdStpActive;
END_REGION

REGION Network 48: **** 8 - Outputs **** Any Production mode active
   // Any Production mode active
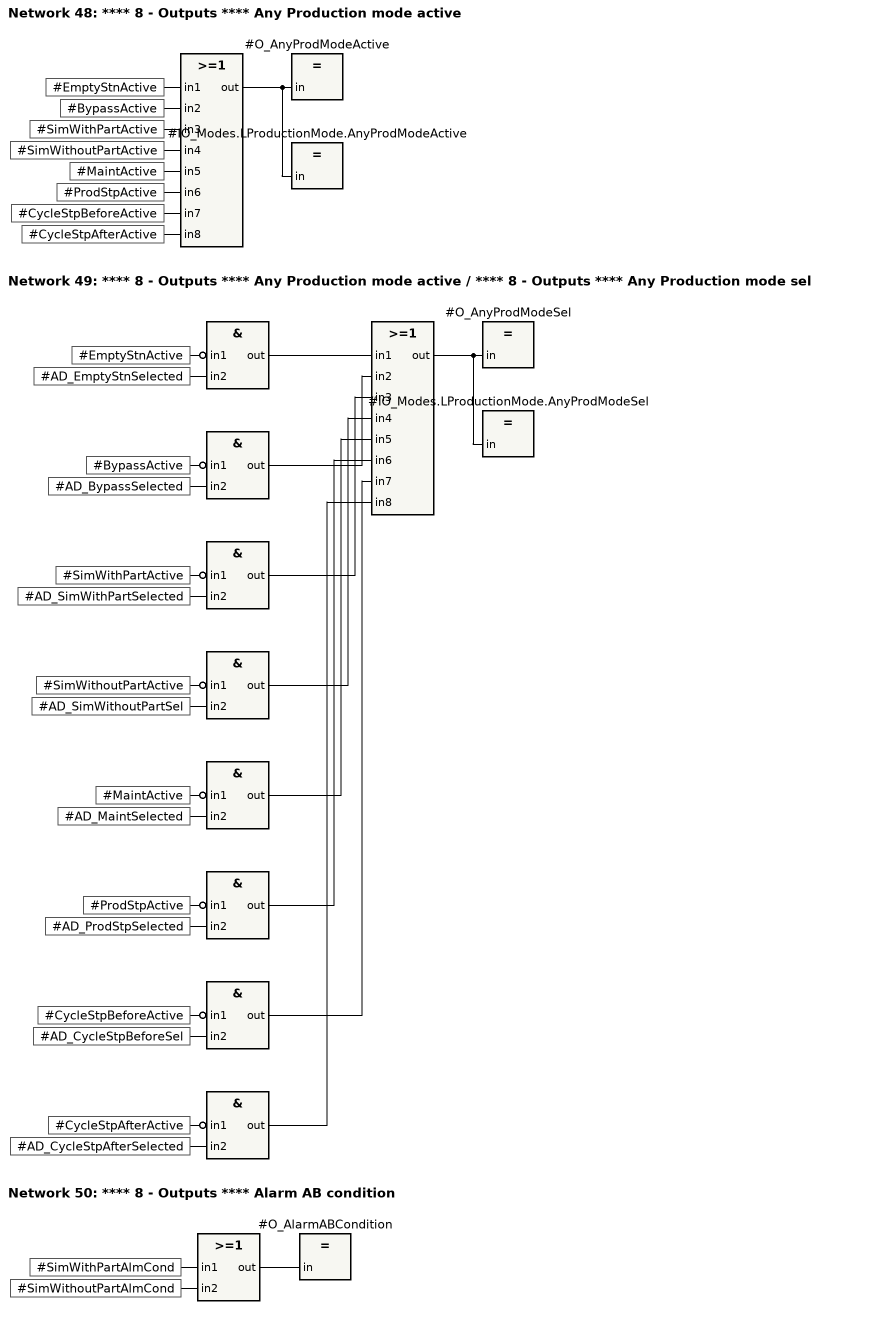
   #O_AnyProdModeActive := #EmptyStnActive OR #BypassActive OR #SimWithPartActive OR #SimWithoutPartActive OR #MaintActive OR #ProdStpActive OR #CycleStpBeforeActive OR #CycleStpAfterActive;
   #IO_Modes.LProductionMode.AnyProdModeActive := #O_AnyProdModeActive;
END_REGION

REGION Network 49: **** 8 - Outputs **** Any Production mode active / **** 8 - Outputs **** Any Production mode sel
   // Any Production mode active
   #O_AnyProdModeSel := (NOT #EmptyStnActive AND #AD_EmptyStnSelected) OR (NOT #BypassActive AND #AD_BypassSelected) OR (NOT #SimWithPartActive AND #AD_SimWithPartSelected) OR (NOT #SimWithoutPartActive AND #AD_SimWithoutPartSel) OR (NOT #MaintActive AND #AD_MaintSelected) OR (NOT #ProdStpActive AND #AD_ProdStpSelected) OR (NOT #CycleStpBeforeActive AND #AD_CycleStpBeforeSel) OR (NOT #CycleStpAfterActive AND #AD_CycleStpAfterSelected);
   #IO_Modes.LProductionMode.AnyProdModeSel := #O_AnyProdModeSel;
END_REGION

REGION Network 50: **** 8 - Outputs **** Alarm AB condition
   // Alarm AB condition
   #O_AlarmABCondition := #SimWithPartAlmCond OR #SimWithoutPartAlmCond;
END_REGION

REGION Network 51: **** 9 - Alarm Summary **** Alarm A
   // Summary of alarms A
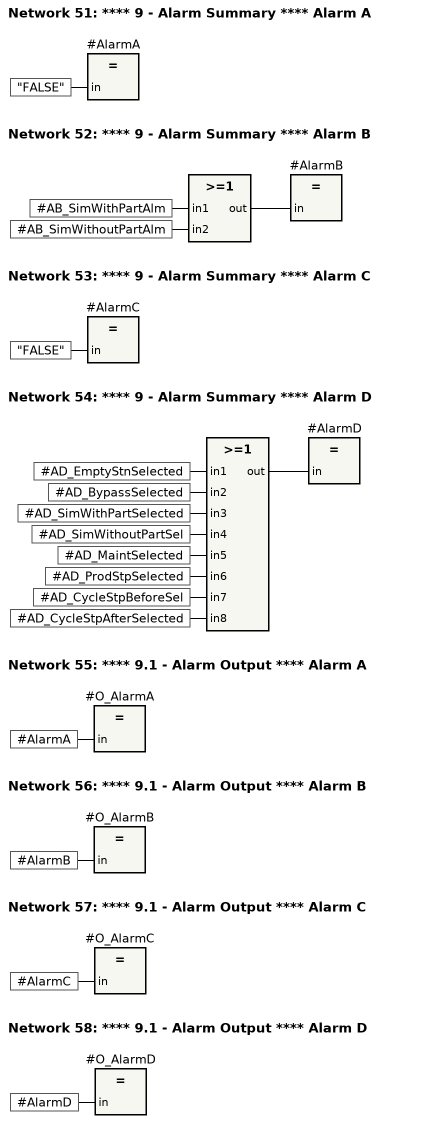
   #AlarmA := "FALSE";
END_REGION

REGION Network 52: **** 9 - Alarm Summary **** Alarm B
   // Summary of alarms B
   #AlarmB := #AB_SimWithPartAlm OR #AB_SimWithoutPartAlm;
END_REGION

REGION Network 53: **** 9 - Alarm Summary **** Alarm C
   // Summary of alarms C
   #AlarmC := "FALSE";
END_REGION

REGION Network 54: **** 9 - Alarm Summary **** Alarm D
   // Summary of alarms D
   #AlarmD := #AD_EmptyStnSelected OR #AD_BypassSelected OR #AD_SimWithPartSelected OR #AD_SimWithoutPartSel OR #AD_MaintSelected OR #AD_ProdStpSelected OR #AD_CycleStpBeforeSel OR #AD_CycleStpAfterSelected;
END_REGION

REGION Network 55: **** 9.1 - Alarm Output **** Alarm A
   // Summary of alarms A
   #O_AlarmA := #AlarmA;
END_REGION

REGION Network 56: **** 9.1 - Alarm Output **** Alarm B
   // Summary of alarms B
   #O_AlarmB := #AlarmB;
END_REGION

REGION Network 57: **** 9.1 - Alarm Output **** Alarm C
   // Summary of alarms C
   #O_AlarmC := #AlarmC;
END_REGION

REGION Network 58: **** 9.1 - Alarm Output **** Alarm D
   // Summary of alarms D
   #O_AlarmD := #AlarmD;
END_REGION

REGION Network 59: **** 9.2 - Alarm DWord**** Alarm To DWord
   // Alarm Word
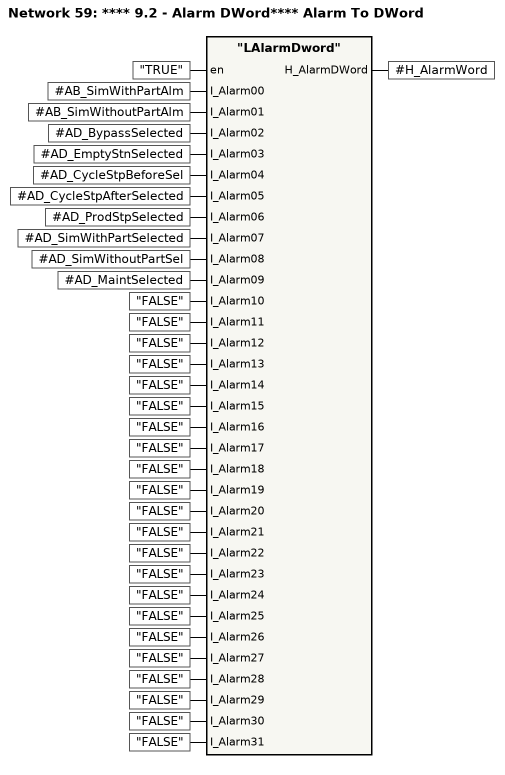
   IF "TRUE" THEN
       "LAlarmDword"(I_Alarm00 := #AB_SimWithPartAlm,
                     I_Alarm01 := #AB_SimWithoutPartAlm,
                     I_Alarm02 := #AD_BypassSelected,
                     I_Alarm03 := #AD_EmptyStnSelected,
                     I_Alarm04 := #AD_CycleStpBeforeSel,
                     I_Alarm05 := #AD_CycleStpAfterSelected,
                     I_Alarm06 := #AD_ProdStpSelected,
                     I_Alarm07 := #AD_SimWithPartSelected,
                     I_Alarm08 := #AD_SimWithoutPartSel,
                     I_Alarm09 := #AD_MaintSelected,
                     I_Alarm10 := "FALSE",
                     I_Alarm11 := "FALSE",
                     I_Alarm12 := "FALSE",
                     I_Alarm13 := "FALSE",
                     I_Alarm14 := "FALSE",
                     I_Alarm15 := "FALSE",
                     I_Alarm16 := "FALSE",
                     I_Alarm17 := "FALSE",
                     I_Alarm18 := "FALSE",
                     I_Alarm19 := "FALSE",
                     I_Alarm20 := "FALSE",
                     I_Alarm21 := "FALSE",
                     I_Alarm22 := "FALSE",
                     I_Alarm23 := "FALSE",
                     I_Alarm24 := "FALSE",
                     I_Alarm25 := "FALSE",
                     I_Alarm26 := "FALSE",
                     I_Alarm27 := "FALSE",
                     I_Alarm28 := "FALSE",
                     I_Alarm29 := "FALSE",
                     I_Alarm30 := "FALSE",
                     I_Alarm31 := "FALSE",
                     H_AlarmDWord => #H_AlarmWord);
   END_IF;
END_REGION
END_FUNCTION_BLOCK
